SUBAPPLICATION Ventilsteuerung_Uebung_043 (* Scaling Function Block with limits Testing *)
  (* Standard: 61499-2 *)
  (* Version 1.0, 2023-10-23, franz *)
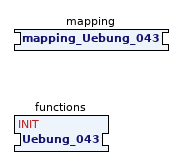
  SUBAPPS
    mapping : mapping_Uebung_043;
    functions : Uebung_043;
  END_SUBAPPS
END_SUBAPPLICATION
